{attribute 'GeneratedUsingTerminal: EL9410-0000-0016'}
{attribute addProperty BoxType "EL9410-0000-0016"}
{attribute addProperty Id "UndervoltageAT %I*BOOL1"}
{attribute addProperty CRC "2984778146"}
{attribute addProperty Size "1"}
TYPE Status_Us_B1E819A2 EXTENDS InputBase_8311D824 :
STRUCT
	{attribute addProperty Name "Undervoltage"}
	Undervoltage AT %I* : BOOL;
END_STRUCT
END_TYPE

(* stored: Version 1.2.0.0, ProductVersion 3.1.4024.11
   DUT Status_Us_B1E819A2: Id {5fab46b7-a7fe-4643-9014-d800725498bf} *)
